{attribute 'qualified_only'}
VAR_GLOBAL
	
		
	{attribute 'OPC.UA.DA' := '1'}
  	{attribute 'OPC.UA.DA.StructuredType' := '1'}
	DTTPOP:	ST_INPUTS_POP;
	
	
	
END_VAR

(* stored: Version 1.1.0.1, ProductVersion 3.1.4024.12
   GVL Inputs: Id {24ddd43c-f29f-4d83-9645-9498c876c4a8} *)
